statusInfoReadyEdge(CLK := NOT getRouterStatusInfo.bBusy AND NOT getRouterStatusInfo.bError);
IF (statusInfoReadyEdge.Q) THEN
	totalMem := DWORD_TO_DINT(statusInfo.maxMem) / IING.ONE_KBYTE;
	freeMem := DWORD_TO_DINT(statusInfo.maxMemAvail) / IING.ONE_KBYTE;
	FC_GetLogger().info(iData := FC_4strConcat(iStr1 := 'Memory usage (KB): ', iStr2 := DINT_TO_STRING(freeMem),
		iStr3 := ' / ', iStr4 := DINT_TO_STRING(totalMem)));
END_IF


// I believe it goes to error in livonia since no data coming from this one, check out and handle errors

END_FUNCTION_BLOCK

// ---- BASE/Misc/FB_OneCycleSignalTof.TcPOU
FUNCTION_BLOCK FB_OneCycleSignalTof		// Delays iSignal by 1 PLC cycle
VAR_INPUT
	iSignal:		BOOL;	// signal to be delayed
END_VAR
VAR_OUTPUT
	oSignal:		BOOL;	// 1 PLC cycle delayed signal
END_VAR
VAR
	fallingEdge:	F_TRIG;
END_VAR

fallingEdge(CLK := iSignal);
oSignal := iSignal OR fallingEdge.Q;

END_FUNCTION_BLOCK

// ---- BASE/Misc/FB_TofOnRtrig.TcPOU
FUNCTION_BLOCK FB_TofOnRtrig		// Monitors a signal (R_TRIG) and creates a TOF
VAR_INPUT
	iBool:		BOOL;	// Signal to be monitored
	iTime:		TIME;	// TOF time
END_VAR
VAR_OUTPUT
	oBool: 		BOOL;	// Set TRUE for iTime on a rising edge of iBool
END_VAR
VAR
	rtrig:		R_TRIG;
	tof:		TOF;
END_VAR

rtrig(CLK := iBool);
tof(IN := rtrig.Q, PT := iTime, Q => oBool);

END_FUNCTION_BLOCK

// ---- BASE/Misc/FC_GetLocalAmsNetId.TcPOU
FUNCTION FC_GetLocalAmsNetId : T_AmsNetId		// Returns the local AMS net id

FC_GetLocalAmsNetId := IING.localAmsNetId;

END_FUNCTION

// ---- BASE/Misc/FC_GetLocalHostName.TcPOU
FUNCTION FC_GetLocalHostName : T_MaxString	// Returns the local host name

FC_GetLocalHostName := IING.localHostName;

END_FUNCTION

// ---- BASE/Misc/FC_GetMax3Arg.TcPOU
FUNCTION FC_GetMax3Arg : REAL
VAR_INPUT
	iVal1:	REAL;
	iVal2:	REAL;
	iVal3:	REAL;
END_VAR
VAR
	maxVal:	REAL;
END_VAR

maxVal := MAX(iVal1, iVal2);
maxVal := MAX(maxVal, iVal3);

FC_GetMax3Arg := maxVal;

END_FUNCTION

// ---- BASE/Misc/FC_GetMax3Lreals.TcPOU
FUNCTION FC_GetMax3Lreals : LREAL		// Returns the maximum of specified values
VAR_INPUT
	iLreal1:	LREAL;
	iLreal2:	LREAL;
	iLreal3:	LREAL;
END_VAR

FC_GetMax3Lreals := MAX(iLreal1, iLreal2);
FC_GetMax3Lreals := MAX(FC_GetMax3Lreals, iLreal3);

END_FUNCTION

// ---- BASE/Misc/FC_GetMax4Arg.TcPOU
FUNCTION FC_GetMax4Arg : REAL
VAR_INPUT
	iVal1:	REAL;
	iVal2:	REAL;
	iVal3:	REAL;
	iVal4:	REAL;
END_VAR
VAR
	maxVal:	REAL;
END_VAR

maxVal := FC_GetMax3Arg(iVal1, iVal2, iVal3);
maxVal := MAX(maxVal, iVal4);

FC_GetMax4Arg := maxVal;

END_FUNCTION

// ---- BASE/Misc/FC_GetMin2Arg.TcPOU
FUNCTION FC_GetMin2Arg : REAL
VAR_INPUT
	iVal1:	REAL;		// Must not be zero
	iVal2:	REAL;
END_VAR
VAR
	minVal:	REAL;
END_VAR

minVal := iVal1;

IF (iVal2 <> 0) THEN
	minVal := MIN(minVal, iVal2);
END_IF

FC_GetMin2Arg := minVal;

END_FUNCTION

// ---- BASE/Misc/FC_GetMin3Arg.TcPOU
FUNCTION FC_GetMin3Arg : REAL
VAR_INPUT
	iVal1:	REAL;		// Must not be zero
	iVal2:	REAL;
	iVal3:	REAL;
END_VAR
VAR
	minVal:	REAL;
END_VAR

minVal := FC_GetMin2Arg(iVal1, iVal2);
minVal := FC_GetMin2Arg(minVal, iVal3);

FC_GetMin3Arg := minVal;

END_FUNCTION

// ---- BASE/Misc/FC_GetMin3Lreals.TcPOU
FUNCTION FC_GetMin3Lreals : LREAL		// Returns the minimum of specified values 
VAR_INPUT
	iLreal1:	LREAL;
	iLreal2:	LREAL;
	iLreal3:	LREAL;
END_VAR

FC_GetMin3Lreals := MIN(iLreal1, iLreal2);
FC_GetMin3Lreals := MIN(FC_GetMin3Lreals, iLreal3);

END_FUNCTION

// ---- BASE/Misc/FC_GetMin4Arg.TcPOU
FUNCTION FC_GetMin4Arg : REAL
VAR_INPUT
	iVal1:	REAL;		// Must not be zero
	iVal2:	REAL;
	iVal3:	REAL;
	iVal4:	REAL;
END_VAR
VAR
	minVal:	REAL;
END_VAR

minVal := FC_GetMin3Arg(iVal1, iVal2, iVal3);
minVal := FC_GetMin2Arg(minVal, iVal4);

FC_GetMin4Arg := minVal;

END_FUNCTION

// ---- BASE/NumberUtils/AddREAL.TcPOU
FUNCTION AddREAL : BOOL				// Increments the given UINT value
VAR_INPUT
	iAdd:	REAL;
END_VAR
VAR_IN_OUT
	ioNum:	REAL;		// Value to increment
END_VAR

ioNum := ioNum + iAdd;

END_FUNCTION

// ---- BASE/NumberUtils/DecINT.TcPOU
FUNCTION DecINT : INT				// Increments the given UINT value
VAR_IN_OUT
	ioNum:	INT;		// Value to increment
END_VAR

DecINT := ioNum := ioNum - 1;

END_FUNCTION

// ---- BASE/NumberUtils/FC_CheckMinMaxInt.TcPOU
FUNCTION FC_CheckMinMaxInt : INT	// Checks if the given value is within the min/max and if not will set either the MIN/MAX value
VAR_INPUT
	iValue:		INT;
	iMin:		INT;
	iMax:		int;
END_VAR

IF (iValue > iMax) THEN
	FC_CheckMinMaxInt := iMax;
ELSIF (iValue < iMin) THEN
	FC_CheckMinMaxInt := iMin;
ELSE
	FC_CheckMinMaxInt := iValue;
END_IF

END_FUNCTION

// ---- BASE/NumberUtils/FC_CheckMinMaxReal.TcPOU
FUNCTION FC_CheckMinMaxReal : REAL		// Checks if the given value is within the min/max and if not will set either the MIN/MAX value
VAR_INPUT
	iValue:		REAL;
	iMin:		REAL;
	iMax:		REAL;
END_VAR

IF (iValue > iMax) THEN
	FC_CheckMinMaxReal := iMax;
ELSIF (iValue < iMin) THEN
	FC_CheckMinMaxReal := iMin;
ELSE
	FC_CheckMinMaxReal := iValue;
END_IF

END_FUNCTION

// ---- BASE/NumberUtils/FC_KeepBetweenMinMax.TcPOU
FUNCTION FC_KeepBetweenMinMax : LREAL			// Keeps the given iValue in between iMin (Floor) and iMax (Ceiling)  
VAR_INPUT
	iValue:		LREAL;
	iMin:		LREAL;
	iMax:		LREAL;
END_VAR

IF (iValue > iMax) THEN
	FC_KeepBetweenMinMax := iMax;
ELSIF (iValue < iMin) THEN
	FC_KeepBetweenMinMax := iMin;
ELSE
	FC_KeepBetweenMinMax := iValue;
END_IF

END_FUNCTION

// ---- BASE/NumberUtils/FC_KeepBetweenMinMaxInt.TcPOU
FUNCTION FC_KeepBetweenMinMaxInt			// Keeps the given ioValue in between iMin (Floor) and iMax (Ceiling)  
VAR_INPUT
	iMin:		INT;
	iMax:		INT;
END_VAR
VAR_IN_OUT
	ioValue:		INT;
END_VAR

IF (ioValue > iMax) THEN
	ioValue := iMax;
ELSIF (ioValue < iMin) THEN
	ioValue := iMin;
END_IF

END_FUNCTION

// ---- BASE/NumberUtils/FC_KeepRealBetweenMinMax.TcPOU
FUNCTION FC_KeepRealBetweenMinMax : REAL			// Keeps the given iValue in between iMin (Floor) and iMax (Ceiling)  
VAR_INPUT
	iValue:		REAL;
	iMin:		REAL;
	iMax:		REAL;
END_VAR

IF (iValue > iMax) THEN
	FC_KeepRealBetweenMinMax := iMax;
ELSIF (iValue < iMin) THEN
	FC_KeepRealBetweenMinMax := iMin;
ELSE
	FC_KeepRealBetweenMinMax := iValue;
END_IF

END_FUNCTION

// ---- BASE/NumberUtils/FC_LimitMaxReal.TcPOU
FUNCTION FC_LimitMaxReal : bool
VAR_INPUT
	iMaster:		REAL;
END_VAR
VAR_IN_OUT
	ioSlave:		REAL;
END_VAR

IF (ioSlave > iMaster) THEN
	ioSlave := iMaster;
END_IF

END_FUNCTION

// ---- BASE/NumberUtils/FC_LimitMinReal.TcPOU
FUNCTION FC_LimitMinReal : bool
VAR_INPUT
	iMaster:	REAL;
END_VAR
VAR_IN_OUT
	ioSlave:		REAL;
END_VAR

IF (ioSlave < iMaster) THEN
	ioSlave := iMaster;
END_IF

END_FUNCTION

// ---- BASE/NumberUtils/FC_WithinMinMax.TcPOU
FUNCTION FC_WithinMinMax : BOOL		// Checks if the specified value is within the target range, returns TRUE if within range, FALSE otherwise
VAR_INPUT
	iValue:			LREAL;		// Value to be checked
	iMin:			LREAL;		// Target value
	iMax:			LREAL;		// This value is allowed below and above
END_VAR

FC_WithinMinMax := (iValue >= iMin) AND (iValue <= iMax);

END_FUNCTION

// ---- BASE/NumberUtils/FC_WithinRange.TcPOU
FUNCTION FC_WithinRange : BOOL		// Checks if the specified value is within the target range, returns TRUE if within range, FALSE otherwise
VAR_INPUT
	iValue:			LREAL;		// Value to be checked
	iTarget:		LREAL;		// Target value
	iRange:			LREAL;		// This value is allowed below and above
END_VAR
VAR
	minValue:	LREAL;
	maxValue:	LREAL;
END_VAR

minValue := iTarget - iRange;
maxValue := iTarget + iRange;
FC_WithinRange := (iValue >= minValue) AND (iValue <= maxValue);

END_FUNCTION

// ---- BASE/NumberUtils/IncINT.TcPOU
FUNCTION IncINT : INT				// Increments the given UINT value
VAR_IN_OUT
	ioNum:	INT;		// Value to increment
END_VAR

IncINT := ioNum := ioNum + 1;

END_FUNCTION

// ---- BASE/NumberUtils/IncUINT.TcPOU
FUNCTION IncUINT : UINT				// Increments the given UINT value
VAR_IN_OUT
	ioNum:	UINT;		// Value to increment
END_VAR

IncUINT := ioNum := ioNum + 1;

END_FUNCTION

// ---- BASE/NumberUtils/IncULINT.TcPOU
FUNCTION IncULINT : ULINT		// Increments the given ULINT value
VAR_IN_OUT
	ioNum:	ULINT;		// Value to increment
END_VAR

IncULINT := ioNum := ioNum + 1;

END_FUNCTION

// ---- BASE/Observer/FB_GenericObserver.TcPOU
FUNCTION_BLOCK ABSTRACT FB_GenericObserver		// To be extended by the REAL observer
VAR
	observers:		ARRAY[0..GVL_GENERIC_OBSERVER.OBSERVER_CNT-1] OF ST_GENERIC_OBSERVER;
	validObservers:	ST_VALID_OBSERVERS;
END_VAR

METHOD PUBLIC deregisterObserver : BOOL
VAR_INPUT
	iWho:				T_SHORT_STR;
END_VAR
VAR
	i: 					INT;
END_VAR
FOR i := 0 TO GVL_GENERIC_OBSERVER.OBSERVER_CNT-1 BY 1 DO
	IF (IsStringEqualIgnoreCase(observers[i].who, iWho)) THEN
		observers[i].who := IING.STRING_BLANK;
	END_IF
END_FOR
END_METHOD

METHOD PUBLIC getObservers : BOOL
VAR_INPUT
END_VAR
VAR
	i: 					INT;
END_VAR
validObservers.cnt := 0;
FOR i := 0 TO GVL_GENERIC_OBSERVER.OBSERVER_CNT-1 BY 1 DO
	IF (FC_StringNotEmpty(observers[i].who)) THEN
		validObservers.observers[validObservers.cnt].observer := observers[i].observer;
		IncInt(validObservers.cnt);
	END_IF
END_FOR
END_METHOD

METHOD PUBLIC registerObserver : BOOL
VAR_INPUT
	iWho:				T_SHORT_STR;
	iObserver:			POINTER TO BYTE;
END_VAR
VAR
	i: 					INT;
END_VAR
// Search if already registered, we do not want to register this twice
FOR i := 0 TO GVL_GENERIC_OBSERVER.OBSERVER_CNT-1 BY 1 DO
	IF (IsStringEqualIgnoreCase(observers[i].who, iWho)) THEN
		observers[i].observer := iObserver;	// Override the observer since it may have changed (re-initialised)
		RETURN;		
	END_IF
END_FOR

// Find 1st free element
FOR i := 0 TO GVL_GENERIC_OBSERVER.OBSERVER_CNT-1 BY 1 DO
	IF (FC_StringEmpty(observers[i].who)) THEN
		observers[i].observer := iObserver;
		observers[i].who := iWho;
		RETURN;		
	END_IF
END_FOR
END_METHOD

END_FUNCTION_BLOCK

// ---- BASE/StringUtils/IsStringEqualIgnoreCase.TcPOU
FUNCTION IsStringEqualIgnoreCase : BOOL
VAR_INPUT
	iString1:	STRING;
	iString2:	STRING;
END_VAR

IsStringEqualIgnoreCase := F_ToUCase(iString1) = F_ToUCase(iString2);

END_FUNCTION

// ---- BASE/StringUtils/FC_5strConcat.TcPOU
FUNCTION FC_5strConcat : T_DEFAULT_STR		// Concatenates 4 strings
VAR_INPUT
	iStr1:		T_DEFAULT_STR;
	iStr2:		T_DEFAULT_STR;
	iStr3:		T_DEFAULT_STR;
	iStr4:		T_DEFAULT_STR;
	iStr5:		T_DEFAULT_STR;
END_VAR

FC_5strConcat := CONCAT(FC_4strConcat(iStr1, iStr2, iStr3, iStr4),iStr5);

END_FUNCTION

// ---- BASE/StringUtils/FC_6strConcat.TcPOU
FUNCTION FC_6strConcat : T_DEFAULT_STR		// Concatenates 4 strings
VAR_INPUT
	iStr1:		T_DEFAULT_STR;
	iStr2:		T_DEFAULT_STR;
	iStr3:		T_DEFAULT_STR;
	iStr4:		T_DEFAULT_STR;
	iStr5:		T_DEFAULT_STR;
	iStr6:		T_DEFAULT_STR;
END_VAR

FC_6strConcat := CONCAT(FC_5strConcat(iStr1, iStr2, iStr3, iStr4, iStr5), iStr6);

END_FUNCTION

// ---- BASE/StringUtils/FC_6strConcatSeparator.TcPOU
FUNCTION FC_6strConcatSeparator : T_DEFAULT_STR		// Concatenates 5 strings with given separator
VAR_INPUT
	iSeparator:		STRING := IING.STRING_UNDERSCORE;
	iStr1:			T_DEFAULT_STR;
	iStr2:			T_DEFAULT_STR;
	iStr3:			T_DEFAULT_STR;
	iStr4:			T_DEFAULT_STR;
	iStr5:			T_DEFAULT_STR;
	iStr6:			T_DEFAULT_STR;
END_VAR

FC_6strConcatSeparator := FC_2strConcatSeparator(iSeparator := iSeparator,
	iStr1 := FC_5strConcatSeparator(iSeparator := iSeparator, iStr1 := iStr1, iStr2 := iStr2, iStr3 := iStr3, iStr4 := iStr4, iStr5 := iStr5), iStr2 := iStr6);

END_FUNCTION

// ---- BASE/StringUtils/FC_7strConcat.TcPOU
FUNCTION FC_7strConcat : T_DEFAULT_STR
VAR_INPUT
	iStr1:		T_DEFAULT_STR;
	iStr2:		T_DEFAULT_STR;
	iStr3:		T_DEFAULT_STR;
	iStr4:		T_DEFAULT_STR;
	iStr5:		T_DEFAULT_STR;
	iStr6:		T_DEFAULT_STR;
	iStr7:		T_DEFAULT_STR;
END_VAR

FC_7strConcat := CONCAT(FC_6strConcat(iStr1, iStr2, iStr3, iStr4, iStr5, iStr6), iStr7);

END_FUNCTION

// ---- BASE/StringUtils/FC_7strConcatSeparator.TcPOU
FUNCTION FC_7strConcatSeparator : T_DEFAULT_STR
VAR_INPUT
	iSeparator:		STRING := IING.STRING_UNDERSCORE;
	iStr1:			T_DEFAULT_STR;
	iStr2:			T_DEFAULT_STR;
	iStr3:			T_DEFAULT_STR;
	iStr4:			T_DEFAULT_STR;
	iStr5:			T_DEFAULT_STR;
	iStr6:			T_DEFAULT_STR;
	iStr7:			T_DEFAULT_STR;
END_VAR

FC_7strConcatSeparator := FC_2strConcatSeparator(iSeparator, FC_6strConcatSeparator(iSeparator, iStr1, iStr2, iStr3, iStr4, iStr5, iStr6), iStr7);

END_FUNCTION

// ---- BASE/StringUtils/FC_8strConcat.TcPOU
FUNCTION FC_8strConcat : T_DEFAULT_STR		// Concatenates 4 strings
VAR_INPUT
	iStr1:		T_DEFAULT_STR;
	iStr2:		T_DEFAULT_STR;
	iStr3:		T_DEFAULT_STR;
	iStr4:		T_DEFAULT_STR;
	iStr5:		T_DEFAULT_STR;
	iStr6:		T_DEFAULT_STR;
	iStr7:		T_DEFAULT_STR;
	iStr8:		T_DEFAULT_STR;
END_VAR

FC_8strConcat := CONCAT(FC_7strConcat(iStr1, iStr2, iStr3, iStr4, iStr5, iStr6, iStr7), iStr8);

END_FUNCTION

// ---- BASE/StringUtils/FC_8strConcatSeparator.TcPOU
FUNCTION FC_8strConcatSeparator : T_DEFAULT_STR
VAR_INPUT
	iSeparator:		STRING := IING.STRING_UNDERSCORE;
	iStr1:			T_DEFAULT_STR;
	iStr2:			T_DEFAULT_STR;
	iStr3:			T_DEFAULT_STR;
	iStr4:			T_DEFAULT_STR;
	iStr5:			T_DEFAULT_STR;
	iStr6:			T_DEFAULT_STR;
	iStr7:			T_DEFAULT_STR;
	iStr8:			T_DEFAULT_STR;
END_VAR

FC_8strConcatSeparator := FC_2strConcatSeparator(iSeparator, FC_7strConcatSeparator(iSeparator, iStr1, iStr2, iStr3, iStr4, iStr5, iStr6, iStr7), iStr8);

END_FUNCTION

// ---- BASE/StringUtils/FC_FindLastOccurence.TcPOU
FUNCTION FC_FindLastOccurence : INT		// Finds the last occurance of a character inside a string
VAR_INPUT
	iStr:			T_MaxString;		// String in where to search
	iStrTofind:		T_SHORT_STR;		// Character to search for
END_VAR
VAR
	i:			INT;
	pos:		INT;
	str:		T_MaxString;
	strLen:		INT;
END_VAR

// Example
// C:\Users\Administrator\Desktop\restartHmi.bat
//   3     9             23      31

FC_FindLastOccurence := 0;
str := iStr;
pos := FIND(str, iStrTofind);
WHILE (pos > 0)  DO
	strLen := LEN(str);
	pos := FIND(str, iStrTofind);
	str := MID(STR := str, LEN := strLen - pos, POS := pos + 1);
	FC_FindLastOccurence := FC_FindLastOccurence + pos;
END_WHILE

END_FUNCTION

// ---- BASE/StringUtils/FC_InitializeNameAsNeeded.TcPOU
FUNCTION FC_InitializeNameAsNeeded	// Can be used to initialize the given name of a component
VAR_INPUT
	iInit:	T_SHORT_STR;		// Initial value
END_VAR
VAR_IN_OUT
	ioMonitor:	T_SHORT_STR;	// String to be monitored
END_VAR

IF (NOT FC_IsBaseNameDefined(ioMonitor)) THEN
	ioMonitor := iInit;
END_IF

END_FUNCTION

// ---- BASE/StringUtils/FC_IsBaseNameDefined.TcPOU
FUNCTION FC_IsBaseNameDefined : bool
VAR_INPUT
	iName:	STRING;
END_VAR
VAR
	equalsNameHere:			BOOL;
	equalsQuestionMarks:	BOOL;
END_VAR

equalsQuestionMarks := IsStringEqualIgnoreCase(iName, IING.STRING_BASE_SETTINGS_INITIAL_NAME);
equalsNameHere := IsStringEqualIgnoreCase(iName, 'name here');

FC_IsBaseNameDefined := NOT equalsQuestionMarks AND NOT equalsNameHere AND FC_StringNotEmpty(iName);

END_FUNCTION

// ---- BASE/StringUtils/FC_LrealFormatter.TcPOU
FUNCTION FC_LrealFormatter : T_SHORT_STR
VAR_INPUT
	iLreal:				LREAL;
	iNumberOfDecimals:	INT;
END_VAR

FC_LrealFormatter := LREAL_TO_FMTSTR(in := iLreal, iPrecision := iNumberOfDecimals, bRound := FALSE);

END_FUNCTION

// ---- BASE/StringUtils/FC_RealFormatter.TcPOU
FUNCTION FC_RealFormatter : T_SHORT_STR
VAR_INPUT
	iReal:				REAL;
	iNumberOfDecimals:	INT;
END_VAR

FC_RealFormatter := LREAL_TO_FMTSTR(in := iReal, iPrecision := iNumberOfDecimals, bRound := FALSE);

END_FUNCTION

// ---- LOGGING/FileLogger/FB_FileLogger.TcPOU
FUNCTION_BLOCK FB_FileLogger IMPLEMENTS I_Logger				// File logger implementation
VAR_INPUT
	iAmsNetId:					T_AmsNetId := IING.STRING_BLANK;	// Where to write the file
	iPath:						T_DEFAULT_STR;					// Path where to log, this MAY NOT contain the file name
	iFileName:					T_SHORT_STR;					// File name for the log files, US style date will be prepended to the file name
END_VAR
VAR_OUTPUT
	oHmi:						ST_FILE_LOGGER_HMI;
END_VAR
VAR
	tcHmiCs:	TC_HMI_CS;	


	service:					ST_FILE_LOGGER_SERVICE;
	controlSignalsFb:			FB_ControlSignalsV2;
	
	
	currentFileNameAndPath:		FB_FileNameAndPath;
	fileWriter:					FB_FileWriterV2;
	
	stopWriting:				BOOL;							// Needed to we can rename the file
	fileScanner:				FB_FileScannerV2;
	higestNumberInFileName:		INT;
	
	newFileName:				T_SHORT_STR;
	newFileNameHelper:			FB_FileNameAndPath;
	fileRenamer:				FB_FileRename;
	fileRenameError:			UDINT;
	lastFileSize:				DINT;
	autoResetTimer:				TON;
	tracingTimer:				TON;
	
	stepChanged:				BOOL;
	step:						E_FILE_LOGGER_STEPS;
	oldStepForStepChangeOnly:	E_FILE_LOGGER_STEPS;			// Dont use for anything else
	prevStep:					E_FILE_LOGGER_STEPS;
	
	observerName:				STRING := 'fileLogger';
END_VAR
VAR PERSISTENT
	settings:					ST_FILE_LOGGER_SETTINGS;
	fileCnt:					INT := 0;
	initCalled:	 				INT;
	reInitCalled:				INT;
	exitCalled:					INT;
END_VAR

controlSignalsFb(iExternalReset := autoResetTimer.Q, ioTcHmi := tcHmiCs);
currentFileNameAndPath.setPathAndFileName(iPath := iPath, iFileName := FC_2strConcatSeparator(iSeparator := IING.STRING_UNDERSCORE, iStr1 := FC_GetUsDateString(), iStr2 := iFileName));

CASE step OF
	E_FILE_LOGGER_STEPS.WAIT_ACTIVITY:
		// When the file gets renamed, the fileSize from the writer gets updated ONLY after the next file write, here we ensure we dont start renaming instantly after the previous rename  
		gotoNextStep(iCondition := fileWriter.oFileSize <> lastFileSize, iNextStep := E_FILE_LOGGER_STEPS.CHECK_SIZE);
	
	E_FILE_LOGGER_STEPS.CHECK_SIZE:
		gotoNextStep(iCondition := (fileWriter.oFileSize > settings.MaxFileSizeMB * IING.ONE_MBYTE), iNextStep := E_FILE_LOGGER_STEPS.CLOSE_FILE);
	
	E_FILE_LOGGER_STEPS.CLOSE_FILE:
		gotoNextStep(iCondition := fileWriter.oFileClosed, iNextStep := E_FILE_LOGGER_STEPS.SCAN_FOLDER);
	
	E_FILE_LOGGER_STEPS.SCAN_FOLDER:
		gotoNextStep(iCondition := fileScanner.oDone, iNextStep := E_FILE_LOGGER_STEPS.ITERATE_FILES);
	
	E_FILE_LOGGER_STEPS.ITERATE_FILES:
		higestNumberInFileName := iterateFiles(iBaseName := currentFileNameAndPath.getFileNameWithExtension(),
			iScannedFiles := ADR(fileScanner.oFiles), iNumberOfFiles := fileScanner.oFilesFound);
	
		gotoNextStep(iCondition := TRUE, iNextStep := E_FILE_LOGGER_STEPS.RENAME_FILE);

	E_FILE_LOGGER_STEPS.RENAME_FILE:
		gotoNextStep(iCondition := fileRenamer.bError, iNextStep := E_FILE_LOGGER_STEPS.RENAME_FILE_ERROR);
		gotoNextStep(iCondition := NOT fileRenamer.bBusy, iNextStep := E_FILE_LOGGER_STEPS.WAIT_ACTIVITY);
		
	E_FILE_LOGGER_STEPS.RENAME_FILE_ERROR:
		gotoNextStep(iCondition := controlSignalsFb.oControlSignals^.out.resetPulse, iNextStep := E_FILE_LOGGER_STEPS.CHECK_SIZE);
ELSE
	step := E_FILE_LOGGER_STEPS.WAIT_ACTIVITY;
END_CASE
updateOldStep();

// For rename to succeed, the log file is first to be closed, when rename fails, we let the logging continue hence that step is not included here
// One thing to notice is that when doLog is called while file rename is ongoing, the file writer will automatically buffer the data and write to file as soon as renaming is completed
stopWriting := (step = E_FILE_LOGGER_STEPS.CLOSE_FILE) OR (step = E_FILE_LOGGER_STEPS.SCAN_FOLDER) OR (step = E_FILE_LOGGER_STEPS.ITERATE_FILES) OR (step = E_FILE_LOGGER_STEPS.RENAME_FILE);

fileWriter(iKeepFileOpen := TRUE, iAmsNetId := iAmsNetId, iFileNameAndPath := currentFileNameAndPath.getFileNameAndPath(), iFlush := service.doFileFlush, iStopWriting := stopWriting,
	iControlSignals := controlSignalsFb.oControlSignals^.out, oFileWriterRecordCnt => oHmi.fileWriterRecordCnt, oFileWriterBytesUsed => oHmi.fileWriterBytesUsed);

fileScanner(iAmsNetId := iAmsNetId, iPath := iPath, iFileName := currentFileNameAndPath.getFileNameWithExtension(),
	iScan := (step = E_FILE_LOGGER_STEPS.SCAN_FOLDER) OR (step = E_FILE_LOGGER_STEPS.ITERATE_FILES), iControlSignals := controlSignalsFb.oControlSignals^.out);

IF (stepChanged AND (step = (E_FILE_LOGGER_STEPS.RENAME_FILE))) THEN
	lastFileSize := fileWriter.oFileSize;
	newFileName := CONCAT(STR1 := currentFileNameAndPath.getFileNameNoExtension(), STR2 := INT_TO_STRING(higestNumberInFileName + 1));
	newFileNameHelper.setPath_FileNameAndExtension(iPath := iPath, iFileName := newFileName, iExtension := currentFileNameAndPath.getExtension());
END_IF	

fileRenamer(sNetId := iAmsNetId, sOldName := currentFileNameAndPath.getFileNameAndPath(), sNewName := newFileNameHelper.getFileNameAndPath(), ePath := E_OpenPath.PATH_GENERIC,
	bExecute := (step = E_FILE_LOGGER_STEPS.RENAME_FILE), tTimeout := IING.ADS_WRITE_TIMEOUT, nErrID => fileRenameError);

autoSwitchOffTracing();
autoReset();
hmi();

METHOD autoReset : BOOL
autoResetTimer(IN := oHmi.error, PT := settings.autoResetTime);
END_METHOD

METHOD PRIVATE autoSwitchOffTracing : BOOL	// Tracing can create a lot of file writing and load, therefore we switch this off after a while
oHmi.tracingOn := settings.logLevel = E_LOG_LEVEL.TRACE;

tracingTimer(IN := settings.enableMaxTracingTime AND oHmi.tracingOn, PT := settings.maxTracingTime, ET => oHmi.tracingTimeExpired);
IF (tracingTimer.Q) THEN
	settings.logLevel := E_LOG_LEVEL.ERROR;
END_IF
END_METHOD

METHOD PUBLIC debug : BOOL	// Logs the data with log level 'DEBUG'
VAR_INPUT
	iData:		T_DEFAULT_STR;						// Data to be logged, limited to 255 characters
END_VAR
doLog(iData := iData, iLevel := E_LOG_LEVEL.DEBUG);
END_METHOD

METHOD PUBLIC deregister : BOOL
VAR_INPUT
	iWho:				T_SHORT_STR;
END_VAR
END_METHOD

METHOD PUBLIC doLog : BOOL		// Logs the data to the file (depending on the activated log level)
								// Timestamp is always added in front of the data
VAR_INPUT
	iData:					T_DEFAULT_STR;						// Data to be logged, limited to 255 characters
	iLevel:					E_LOG_LEVEL := E_LOG_LEVEL.ERROR;	// Log level
END_VAR
VAR
	logLevel:				FB_LogLevel;
	header:					T_DEFAULT_STR;
	fullLine:				T_LONG_STR_512;
	
	runningNumberAsString:	T_SHORT_STR;
	eventIdAsString:		T_SHORT_STR;
	
	testSuccess: 			BOOL;
END_VAR
(*
v: Visible
						doLog called with
						-----------------
						ERROR		WARN		INFO		DEBUG		TRACE
Current log level
-----------------
OFF						
ERROR					v
WARN					v			v
INFO					v			v			v
DEBUG					v			v			v			v
TRACE					v			v			v			v			v
*)

// Logging is only done when the log level is higher or equal the current log level
IF (iLevel >= settings.logLevel) THEN
	logLevel.set(iLevel);

	header := FC_2strConcatSeparator (iSeparator := IING.STRING_SPACE, iStr1 := FC_GetLocalDateAndTimeString(), iStr2 := logLevel.asString());
	
	
	// iData can be up to 255 chars, including the header therefore more than 255, we use CONCAT2 and 'long' string 
	fullLine := CONCAT(STR1 := header, STR2 := IING.STRING_SPACE);
	testSuccess := CONCAT2(pSrcString1  := ADR(fullLine), pSrcString2 := ADR(iData), pDstString := ADR(fullLine), nDstSize := SIZEOF(fullLine));
	testSuccess := CONCAT2(pSrcString1  := ADR(fullLine), pSrcString2 := ADR(IING.STRING_LINE_FEED), pDstString := ADR(fullLine), nDstSize := SIZEOF(fullLine));
	
	fileWriter.doWrite(fullLine);
END_IF

// Just in case something went wrong and the level is not within the enum range
IF (settings.logLevel > E_LOG_LEVEL.OFF) THEN
	settings.logLevel := E_LOG_LEVEL.ERROR;
END_IF
END_METHOD

METHOD PUBLIC error : BOOL	// Logs the data with log level 'ERROR'
VAR_INPUT
	iData:		T_DEFAULT_STR;						// Data to be logged, limited to 255 characters
END_VAR
doLog(iData := iData, iLevel := E_LOG_LEVEL.ERROR);
END_METHOD

METHOD FB_exit : BOOL
VAR_INPUT
	bInCopyCode : BOOL; // if TRUE, the exit method is called for exiting an instance that is copied afterwards (online change).
END_VAR
IncInt(exitCalled);

//FC_GetLogger().deregister(observerName);
END_METHOD

METHOD FB_init : BOOL
VAR_INPUT
	bInitRetains : BOOL; // if TRUE, the retain variables are initialized (warm start / cold start)
	bInCopyCode : BOOL;  // if TRUE, the instance afterwards gets moved into the copy code (online change)
END_VAR
IncInt(initCalled);

//FC_GetLogger().register(observerName, THIS^);
END_METHOD

METHOD FB_reinit : BOOL
IncInt(reInitCalled);

//FC_GetLogger().register(observerName, THIS^);
END_METHOD

METHOD PRIVATE gotoNextStep : BOOL
VAR_INPUT
	iCondition:	BOOL;
	iNextStep:	E_FILE_LOGGER_STEPS;
END_VAR
IF (NOT (step<>oldStepForStepChangeOnly)) THEN
	IF (iCondition) THEN
		step := iNextStep;
	END_IF
END_IF
END_METHOD

METHOD PRIVATE hmi : BOOL
oHmi.service REF= service;
oHmi.settings REF= settings;
oHmi.controlSignals REF= controlSignalsFb.oControlSignals^.in;

IF (step = E_FILE_LOGGER_STEPS.SCAN_FOLDER) THEN
	oHmi.error := fileScanner.oError;
	oHmi.adsErrorCode := fileScanner.oAdsErrorCode;
ELSIF (step = E_FILE_LOGGER_STEPS.RENAME_FILE_ERROR) THEN
	oHmi.error := TRUE;	
	oHmi.adsErrorCode := FC_GetAdsErrorCode(fileRenameError);				
ELSE
	oHmi.error := fileWriter.oError;
	oHmi.adsErrorCode := fileWriter.oAdsErrorCode;
END_IF
	
oHmi.amsNetId := iAmsNetId;
oHmi.fileNameAndPath := currentFileNameAndPath.getFileNameAndPath();

oHmi.fileWriterOverflowCount := fileWriter.oOverflowCount;

// Found from autoSwitchOffTracing
//oHmi.tracingOn 
//oHmi.tracingTimeLeft
END_METHOD

METHOD PUBLIC info : BOOL	// Logs the data with log level 'INFO'
VAR_INPUT
	iData:		T_DEFAULT_STR;						// Data to be logged, limited to 255 characters
END_VAR
doLog(iData := iData, iLevel := E_LOG_LEVEL.INFO);
END_METHOD

METHOD PRIVATE iterateFiles : INT		// Iterates the given files and stores the highest number as appended in the base file name
VAR_INPUT
	iBaseName:				T_SHORT_STR;				// Base name, eg. 2019-11-14-logging
	iScannedFiles:			POINTER TO T_SHORT_STR;		// Array of files as given by FB_FileScanner matching the base name
	iNumberOfFiles:			INT;						// Number of files in the scannedFiles array
END_VAR
VAR 
	i:						INT;						// For loop
	baseNameHelper:			FB_FileNameAndPath;
	scannedFileHelper:		FB_FileNameAndPath;
	fileNumberAsString:		T_SHORT_STR;
	fileNumber:				INT;
END_VAR
// Iterates the given files and stores the highest number as appended in the base file name, in this example it would be 3
// 2019-11-14-logging1.txt
// 2019-11-14-logging2.txt
// 2019-11-14-logging3.txt
baseNameHelper.setPathAndFileName(iPath := iPath, iFileName := iBaseName);

FOR i := 0 TO iNumberOfFiles -1 BY 1 DO
	scannedFileHelper.setPathAndFileName(iPath := iPath, iFileName := iScannedFiles[i]);
	fileNumberAsString := RIGHT(STR := scannedFileHelper.getFileNameNoExtension(), SIZE := LEN(scannedFileHelper.getFileNameNoExtension()) - LEN(baseNameHelper.getFileNameNoExtension()));
	
	fileNumber := STRING_TO_INT(fileNumberAsString);// If this fails, 0 will be returned so this is safe to do
	iterateFiles := MAX(fileNumber, iterateFiles);
END_FOR
END_METHOD

METHOD PUBLIC register : BOOL
VAR_INPUT
	iWho:		T_SHORT_STR;
	iObserver:	I_Logger;
END_VAR
END_METHOD

METHOD PUBLIC trace : BOOL	// Logs the data with log level 'TRACE'
VAR_INPUT
	iData:		T_DEFAULT_STR;						// Data to be logged, limited to 255 characters
END_VAR
doLog(iData := iData, iLevel := E_LOG_LEVEL.TRACE);
END_METHOD

ACTION updateOldStep:
IF (step <> oldStepForStepChangeOnly) THEN
	stepChanged := TRUE;
	prevStep := oldStepForStepChangeOnly;			// Otherwise next SWITCH CASE checks oldStep which was just updated here!!
	oldStepForStepChangeOnly := step;
ELSE 
	stepChanged := FALSE;
END_IF
END_ACTION

METHOD PUBLIC warn : BOOL	// Logs the data with log level 'WARN'
VAR_INPUT
	iData:		T_DEFAULT_STR;						// Data to be logged, limited to 255 characters
END_VAR
doLog(iData := iData, iLevel := E_LOG_LEVEL.WARN);
END_METHOD

END_FUNCTION_BLOCK

// ---- LOGGING/FileLogger/FB_FileNameAndPath.TcPOU
FUNCTION_BLOCK FB_FileNameAndPath		// Utility function for making file path/naming easier
VAR
	path:				T_DEFAULT_STR;
	fileName:			T_DEFAULT_STR;
	extension:			T_SHORT_STR;
	fileNameAndPath:	T_DEFAULT_STR;
END_VAR

METHOD public getExtension : T_SHORT_STR		// Returns the file extension
getExtension := extension;
END_METHOD

METHOD PUBLIC getFileNameAndPath : T_DEFAULT_STR		// Returns the full file name and path (including extension)
getFileNameAndPath := fileNameAndPath;
END_METHOD

METHOD public getFileNameNoExtension : T_DEFAULT_STR		// Returns the file name without the extension
getFileNameNoExtension := fileName;
END_METHOD

METHOD PUBLIC getFileNameWithExtension : T_DEFAULT_STR	// Returns the file name with extension
getFileNameWithExtension := FC_2strConcatSeparator(iSeparator := IING.STRING_DOT, iStr1 := fileName, iStr2 := extension);
END_METHOD

METHOD PUBLIC getPath : T_DEFAULT_STR		// Returns the file path
getPath := path;
END_METHOD

METHOD PUBLIC setPath_FileNameAndExtension : BOOL	// Setter for file name, extension and path
VAR_INPUT
	iPath:			T_DEFAULT_STR;		// Path
	iFileName:		T_SHORT_STR;		// File name excluding the extension
	iExtension:		T_SHORT_STR;		// The file extension
END_VAR
setPathAndFileName(iPath := iPath, iFileName := FC_3strConcat(iStr1 := iFileName, iStr2 := IING.STRING_DOT, iStr3 := iExtension));
END_METHOD

METHOD public setPathAndFileName : BOOL		// Setter for file name (including extension) and path
VAR_INPUT
	iPath:			T_DEFAULT_STR;		// Path
	iFileName:		T_SHORT_STR;		// File name including the extension
END_VAR

VAR
	dotPos:int;
END_VAR
// Construct path having back slash at the end
IF (RIGHT(iPath, 1) = IING.STRING_BACKSLASH) THEN
	path := iPath;
ELSE
	path := CONCAT(iPath, IING.STRING_BACKSLASH);
END_IF

// Construct file name with extension
dotPos := FIND(iFileName, IING.STRING_DOT);
IF (dotPos > 0) THEN
	fileName := LEFT(STR := iFileName, SIZE := dotPos -1);
	extension := RIGHT(STR := iFileName, SIZE := LEN(iFileName) - dotPos);
ELSE
	fileName := iFileName;
	extension := 'missing';
END_IF


fileNameAndPath := CONCAT(path, getFileNameWithExtension());
END_METHOD

END_FUNCTION_BLOCK

// ---- LOGGING/FileLogger/FB_FileWriterV2.TcPOU
FUNCTION_BLOCK FB_FileWriterV2	// Handles writing of lines to a file.  Maximum line length is 256 characters.
VAR_INPUT
	iKeepFileOpen:					BOOL;							// Set TRUE to keep the file open in between writes
	iAmsNetId:						T_AmsNetId := IING.STRING_BLANK;	// Where to write the file
	iFileNameAndPath:				T_DEFAULT_STR;					// File name and path of the file
	iFlush:							BOOL;							// Set TRUE when a file flush is needed (will actually close and re-open the file)
	iStopWriting:					BOOL;							// Used when the caller of this FB wants to temporarily stop writing (eg. when file rename is ongoing)
	iControlSignals:				ST_CONTROL_SIGNALS_OUT;			// Control signals (carrying reset signal)
END_VAR
VAR_OUTPUT
	oFileClosed:					BOOL;
	oFileSize:						DINT;
	oError:							BOOL;							// TRUE if a file writing error occurs
	oAdsErrorCode:					E_ADS_ERRORS;
	oOverflowCount:					UDINT;							// How many times we were not able to write all data to the file (due to internal memory constraints)
	
	oFileWriterRecordCnt:			UDINT;
	oFileWriterBytesUsed:			UDINT;
END_VAR
VAR
	fileHandle:						UINT := 0;
	fileHandleFromFB_FileOpen:		UINT := 0;						// Separate var since overwritten from FB_FileOpen even if not open anymore
	fileOpen:						FB_FileOpen;
	fileWrite:						FB_FileWrite;					// Not using FB_FilePuts since it is limited of writing T_MaxString
	fileClose:						FB_FileClose;

	fileTell:						FB_FileTell;
	
	dataToBeWritten:				BOOL;		// Helper to know when data is buffered and to be written
	
	fileNameCopy:					T_DEFAULT_STR;
	fileNameChangeEdge:				R_TRIG;
	flush:							BOOL;
	
	stepChanged:					BOOL;
	step:							E_FILE_WRITER_STEPS;
	oldStepForStepChangeOnly:		E_FILE_WRITER_STEPS;			// Dont use for anything else
	prevStep:						E_FILE_WRITER_STEPS;
	
	ringBufferMemory:				ARRAY[0..RINGBUFFER_SIZE_IN_BYTES-1] OF BYTE;
	ringBuffer:						FB_MemRingBuffer;
	
	longString:						STRING(LONGSTRING_SIZE_IN_BYTES);	// LEN2 has a restriction to 10000 chars
	
	fileOpeningError:				UDINT;
	fileWritingError:				UDINT;
	fileTellError:					UDINT;
	fileClosingError:				UDINT;
	
	bytesWritten:					UDINT;
END_VAR
VAR PERSISTENT
	overFlowCnt:					UDINT;	// Number of times overflow would have happened
	concatFailure:					UDINT;	// Number of concat failures, should stay at 0
END_VAR
VAR CONSTANT
	RINGBUFFER_SIZE_IN_BYTES:		UDINT := 30000;
	LONGSTRING_SIZE_IN_BYTES:		UDINT := 10000;
END_VAR

// When file name changes (eg. from logger), we need to close and re-open the file (with different name)
fileNameChangeEdge(CLK := NOT (iFileNameAndPath = fileNameCopy));
fileNameCopy := iFileNameAndPath;

IF (fileNameChangeEdge.Q OR iFlush) THEN		// Rising edge can easily get lost while writing is ongoing (can take several PLC cycles), therefore must 'save' it
	flush := TRUE;	
END_IF

dataToBeWritten := ringBuffer.nCount > 0;	// See doWrite

CASE step OF
	E_FILE_WRITER_STEPS.IDLE:
		gotoNextStep(iCondition := NOT iStopWriting AND iKeepFileOpen, iNextStep := E_FILE_WRITER_STEPS.OPEN_FILE);
		gotoNextStep(iCondition := NOT iStopWriting AND NOT iKeepFileOpen AND dataToBeWritten, iNextStep := E_FILE_WRITER_STEPS.OPEN_FILE);
		
	E_FILE_WRITER_STEPS.OPEN_FILE:
		gotoNextStep(iCondition := fileOpen.bError, iNextStep := E_FILE_WRITER_STEPS.OPENING_ERROR);
		gotoNextStep(iCondition := NOT fileOpen.bBusy, iNextStep := E_FILE_WRITER_STEPS.WAIT_DATA);
	
	E_FILE_WRITER_STEPS.WAIT_DATA:
		gotoNextStep(iCondition := dataToBeWritten, iNextStep := E_FILE_WRITER_STEPS.WRITE_LINE);
		gotoNextStep(iCondition := flush OR NOT iKeepFileOpen OR iStopWriting, iNextStep := E_FILE_WRITER_STEPS.CLOSE_FILE);

	E_FILE_WRITER_STEPS.WRITE_LINE:
		gotoNextStep(iCondition := fileWrite.bError, iNextStep := E_FILE_WRITER_STEPS.WRITING_ERROR);
		gotoNextStep(iCondition := NOT fileWrite.bBusy , iNextStep := E_FILE_WRITER_STEPS.CHECK_FILE);
		
	E_FILE_WRITER_STEPS.CHECK_FILE:
		gotoNextStep(iCondition := fileTell.bError, iNextStep := E_FILE_WRITER_STEPS.TELL_ERROR);
		gotoNextStep(iCondition := NOT fileTell.bBusy AND (flush OR iStopWriting OR NOT iKeepFileOpen), iNextStep := E_FILE_WRITER_STEPS.CLOSE_FILE);
		gotoNextStep(iCondition := NOT fileTell.bBusy, iNextStep := E_FILE_WRITER_STEPS.WAIT_DATA);

	E_FILE_WRITER_STEPS.CLOSE_FILE:
		flush := FALSE;
		gotoNextStep(iCondition := fileClose.bError, iNextStep := E_FILE_WRITER_STEPS.CLOSING_ERROR);
		gotoNextStep(iCondition := NOT fileClose.bBusy, iNextStep := E_FILE_WRITER_STEPS.CLEANUP);
	
	E_FILE_WRITER_STEPS.CLEANUP:
		fileHandle := 0;
		gotoNextStep(iCondition := TRUE, iNextStep := E_FILE_WRITER_STEPS.IDLE);
	
	E_FILE_WRITER_STEPS.OPENING_ERROR:
		oAdsErrorCode := FC_GetAdsErrorCode(fileOpeningError);
		gotoNextStep(iCondition := fileHandle <> 0, iNextStep := E_FILE_WRITER_STEPS.CLOSE_FILE);
		gotoNextStep(iCondition := iControlSignals.resetPulse, iNextStep := E_FILE_WRITER_STEPS.IDLE);

	E_FILE_WRITER_STEPS.WRITING_ERROR:
		oAdsErrorCode := FC_GetAdsErrorCode(fileWritingError);
		gotoNextStep(iCondition := fileHandle <> 0, iNextStep := E_FILE_WRITER_STEPS.CLOSE_FILE);
		gotoNextStep(iCondition := iControlSignals.resetPulse, iNextStep := E_FILE_WRITER_STEPS.IDLE);

	E_FILE_WRITER_STEPS.TELL_ERROR:
		oAdsErrorCode := FC_GetAdsErrorCode(fileTellError);
 		gotoNextStep(iCondition := fileHandle <> 0, iNextStep := E_FILE_WRITER_STEPS.CLOSE_FILE);
		gotoNextStep(iCondition := iControlSignals.resetPulse, iNextStep := E_FILE_WRITER_STEPS.IDLE);
		
	E_FILE_WRITER_STEPS.CLOSING_ERROR:
		oAdsErrorCode := FC_GetAdsErrorCode(fileClosingError);
		gotoNextStep(iCondition := iControlSignals.resetPulse, iNextStep := E_FILE_WRITER_STEPS.IDLE);
ELSE
	step := E_FILE_WRITER_STEPS.IDLE;
END_CASE
updateOldStep();


IF (stepChanged AND (step = E_FILE_WRITER_STEPS.WAIT_DATA) AND (prevStep = E_FILE_WRITER_STEPS.OPEN_FILE)) THEN
	fileHandle := fileHandleFromFB_FileOpen;
END_IF

fileOpen(sNetId := iAmsNetId, sPathName := iFileNameAndPath, nMode := FOPEN_MODEAPPEND,
	ePath := PATH_GENERIC, bExecute := (step = E_FILE_WRITER_STEPS.OPEN_FILE), hFile => fileHandleFromFB_FileOpen, tTimeout := IING.ADS_WRITE_TIMEOUT, nErrID => fileOpeningError);
	
// The data must be updated before the writing starts
concatBuffers(stepChanged AND (step = E_FILE_WRITER_STEPS.WRITE_LINE));	// Concatenates all data into a long string so writing is more efficient

fileWrite(sNetId := iAmsNetId, hFile := fileHandle, pWriteBuff := ADR(longString), cbWriteLen := LEN2(ADR(longString)), bExecute := (step = (E_FILE_WRITER_STEPS.WRITE_LINE)),
	tTimeout := IING.ADS_WRITE_TIMEOUT, nErrId => fileWritingError, cbWrite => bytesWritten);
	
fileTell(sNetId := iAmsNetId, hFile := fileHandle, bExecute := (step = E_FILE_WRITER_STEPS.CHECK_FILE), tTimeout := IING.ADS_WRITE_TIMEOUT, nSeekPos => oFileSize,
	nErrId => fileTellError);	
	
fileClose(sNetId := iAmsNetId, hFile := fileHandle, bExecute := (step = (E_FILE_WRITER_STEPS.CLOSE_FILE)), tTimeout := IING.ADS_WRITE_TIMEOUT, nErrId => fileClosingError);

ringBuffer(nCount => oFileWriterRecordCnt, cbSize => oFileWriterBytesUsed);

oFileClosed := (step = E_FILE_WRITER_STEPS.IDLE);		// In idle we can be sure the file is closed
oError := (step = E_FILE_WRITER_STEPS.OPENING_ERROR) OR (step = E_FILE_WRITER_STEPS.WRITING_ERROR) OR (step = E_FILE_WRITER_STEPS.CLOSING_ERROR);
oOverflowCount := overFlowCnt;

IF (iControlSignals.hardResetPulse) THEN
	step := E_FILE_WRITER_STEPS.IDLE;
	ringBuffer.A_Reset();
	flush := FALSE;
END_IF

METHOD PRIVATE concatBuffers : BOOL
VAR_INPUT
	iCondition:			BOOL;
END_VAR
VAR
	bufferedLine:		T_LONG_STR_512;	// Data read back from the ringBuffer, must be as big as iData in the doWrite method!
	trash:				T_LONG_STR_512;	// Must be as big as iData in the doWrite method!
	shouldFit:			BOOL;
	
	bufferedLineLen:	UDINT;
	longStringLen:		UDINT;
END_VAR
IF (iCondition) THEN
	longString := '';
	shouldFit := TRUE;
	WHILE (ringBuffer.nCount > 0 AND shouldFit) DO
		// We get the data but dont delete it yet
		ringBuffer.A_GetHead(pRead := ADR(bufferedLine), cbRead := SIZEOF(bufferedLine), pBuffer := ADR(ringBufferMemory), cbBuffer	:= SIZEOF(ringBufferMemory));

		// Check if bufferedLine will fit to longString
		bufferedLineLen := LEN2(ADR(bufferedLine));
		longStringLen:= LEN2(ADR(longString));
		shouldFit := (longStringLen + bufferedLineLen <= LONGSTRING_SIZE_IN_BYTES);	// Same size as longString
		IF (shouldFit) THEN
			// Here we concat onto longString, this should always succeed
			// If data would be too big for CONCAT2, that data that fits would be added and the rest discarded, therefore we check before hand to ensure all data gets logged correctly
			shouldFit := CONCAT2(pSrcString1  := ADR(longString), pSrcString2 := ADR(bufferedLine), pDstString := ADR(longString), nDstSize := SIZEOF(longString));
			IF (shouldFit) THEN
				// When the data did fit, we remove it from the ringBuffer (we read into a trash variable)
				ringBuffer.A_RemoveHead(pRead := ADR(trash), cbRead := SIZEOF(trash), pBuffer := ADR(ringBufferMemory), cbBuffer	:= SIZEOF(ringBufferMemory));
			ELSE
				// Should never come here
				IncUDINT(concatFailure); 
			END_IF
		ELSE
			;	// Its ok to leave the while loop since we will write (to file) all we got into longString, after that we create another longString and write again
			// The 10000 limitation means our file write, writes mostly 10000 bytes at a time
		END_IF
	END_WHILE
END_IF
END_METHOD

METHOD PUBLIC doWrite : BOOL		// Will add this data to the queue that will be written in the current PLC cycle.  Data is buffered and file write happens at most once/PLC cycle.
VAR_INPUT
	iData:		T_LONG_STR_512;		// The data to be written, up to 512 chars
END_VAR
// Add data to the FIFO

// If SIZEOF is used on iData, the ringbuffer always has entries that are as big as iData, even though the string would be 1 char only
// When using, LEN2, we can fit more data to the ringbuffer since rarely the iData will be the max length
// +1 is to account for the string variables final null (it is required!)
ringBuffer.A_AddTail(pWrite := ADR(iData), cbWrite := (LEN2(ADR(iData)) + 1), 							// What to write
					 pBuffer := ADR(ringBufferMemory), cbBuffer := SIZEOF(ringBufferMemory));	// The ringbuffer's memory	
					 
// If data doesnt fit anymore, bOk will be FALSE					 
IF (NOT ringBuffer.bOk) THEN
	IncUDINT(overflowCnt);	// More data is to be written in this PLC cycle but it doesnt fit the ringBuffer
END_IF
END_METHOD

METHOD PRIVATE gotoNextStep : BOOL
VAR_INPUT
	iCondition:	BOOL;
	iNextStep:	E_FILE_WRITER_STEPS;
END_VAR
IF (NOT (step<>oldStepForStepChangeOnly)) THEN
	IF (iCondition) THEN
		step := iNextStep;
	END_IF
END_IF
END_METHOD

ACTION updateOldStep:
IF (step <> oldStepForStepChangeOnly) THEN
	stepChanged := TRUE;
	prevStep := oldStepForStepChangeOnly;			// Otherwise next SWITCH CASE checks oldStep which was just updated here!!
	oldStepForStepChangeOnly := step;
ELSE 
	stepChanged := FALSE;
END_IF
END_ACTION

END_FUNCTION_BLOCK

// ---- LOGGING/FileLogger/FB_FileScannerV2.TcPOU
FUNCTION_BLOCK FB_FileScannerV2	// Scans the given folder for files with given name
VAR_INPUT
	iAmsNetId:					T_AmsNetId := IING.STRING_BLANK;	// Where to scan for files
	iPath:						T_DEFAULT_STR;					// Path where to scan, this MAY NOT contain the file name
	iFileName:					T_SHORT_STR;					// File names to match, do not include wildcards here
	iScan:						BOOL;							// TRUE will start the scanning
	iControlSignals:			ST_CONTROL_SIGNALS_OUT;			// Control signals (carrying reset signal)
END_VAR
VAR_OUTPUT
	oDone:						BOOL;									// Set TRUE when scanning is completed
	oFiles:						ARRAY[0..MAX_FILES-1] OF T_SHORT_STR;	// List of scanned files matching the given fileName
	oFilesFound:				INT;									// Number of matching files
	oError:						BOOL;									// Set TRUE when a scan error occurs
	oAdsErrorCode:				E_ADS_ERRORS;							// The error code in case oError is TRUE
END_VAR
VAR
	fileNameAndPath:			FB_FileNameAndPath;
	fileCnt:					INT;
	fileToSearch:				T_DEFAULT_STR;
	scanCommand:				E_EnumCmdType;
	scanFolder:					FB_EnumFindFileEntry;
	scanFolderError:			UDINT;

	stepChanged:				BOOL;
	step:						E_FILE_SCANNER_STEPS;
	oldStepForStepChangeOnly:	E_FILE_SCANNER_STEPS;			// Dont use for anything else
	prevStep:					E_FILE_SCANNER_STEPS;
END_VAR
VAR CONSTANT
	MAX_FILES:					INT := 100;
END_VAR

CASE step OF
	E_FILE_SCANNER_STEPS.IDLE:
		gotoNextStep(iCondition := iScan, iNextStep := E_FILE_SCANNER_STEPS.SCAN);
	
	E_FILE_SCANNER_STEPS.SCAN:
		gotoNextStep(iCondition := scanFolder.bError, iNextStep := E_FILE_SCANNER_STEPS.ERROR);
		gotoNextStep(iCondition := NOT scanFolder.bBusy, iNextStep := E_FILE_SCANNER_STEPS.STORE_FILE);	

	E_FILE_SCANNER_STEPS.STORE_FILE:
		IF (NOT scanFolder.bEOE) THEN
			IF (fileCnt < MAX_FILES) THEN
				oFiles[fileCnt] := scanFolder.stFindFile.sFileName;
				IncINT(fileCnt);
			END_IF
			gotoNextStep(iCondition := TRUE, iNextStep := E_FILE_SCANNER_STEPS.SCAN);		
		ELSE
			gotoNextStep(iCondition := TRUE, iNextStep := E_FILE_SCANNER_STEPS.DONE);		
		END_IF	
		
	E_FILE_SCANNER_STEPS.DONE:
		gotoNextStep(iCondition := NOT iScan, iNextStep := E_FILE_SCANNER_STEPS.IDLE);

	E_FILE_SCANNER_STEPS.ERROR:
		oAdsErrorCode := FC_GetAdsErrorCode(scanFolderError);
		gotoNextStep(iCondition := iControlSignals.resetPulse, iNextStep := E_FILE_SCANNER_STEPS.IDLE);
ELSE
	step := E_FILE_SCANNER_STEPS.IDLE;
END_CASE
updateOldStep();


IF (stepChanged AND (step = E_FILE_SCANNER_STEPS.IDLE)) THEN
	fileCnt := 0;
	MEMSET(destAddr := ADR(oFiles), fillByte := 0, SIZEOF(oFiles));
END_IF

IF (stepChanged AND (step = E_FILE_SCANNER_STEPS.SCAN)) THEN
	fileNameAndPath.setPathAndFileName(iPath := iPath, iFileName := iFileName);
	IF (prevStep = E_FILE_SCANNER_STEPS.IDLE) THEN
		fileToSearch := fileNameAndPath.getFileNameNoExtension();

		// Wildcards to find files with similar name
		fileToSearch := FC_3strConcat(iStr1 := fileNameAndPath.getPath(), iStr2 := fileToSearch, iStr3 := IING.STRING_STAR);

		// First scan starts from the beginning (FB_EnumFindFileEntry)
		scanCommand := E_EnumCmdType.eEnumCmd_First;
	ELSE
		// Next scan just continues (FB_EnumFindFileEntry)
		scanCommand := E_EnumCmdType.eEnumCmd_Next;
	END_IF
END_IF

scanFolder(sNetID := iAmsNetId, sPathName := fileToSearch, eCmd := scanCommand, bExecute := (step = E_FILE_SCANNER_STEPS.SCAN), tTimeout := IING.ADS_WRITE_TIMEOUT,
	nErrID => scanFolderError);

oDone := (step = E_FILE_SCANNER_STEPS.DONE);
oFilesFound := fileCnt;
oError := (step = E_FILE_SCANNER_STEPS.ERROR);

METHOD PRIVATE gotoNextStep : BOOL
VAR_INPUT
	iCondition:	BOOL;
	iNextStep:	E_FILE_SCANNER_STEPS;
END_VAR
IF (NOT (step<>oldStepForStepChangeOnly)) THEN
	IF (iCondition) THEN
		step := iNextStep;
	END_IF
END_IF
END_METHOD

ACTION updateOldStep:
IF (step <> oldStepForStepChangeOnly) THEN
	stepChanged := TRUE;
	prevStep := oldStepForStepChangeOnly;			// Otherwise next SWITCH CASE checks oldStep which was just updated here!!
	oldStepForStepChangeOnly := step;
ELSE 
	stepChanged := FALSE;
END_IF
END_ACTION

END_FUNCTION_BLOCK

// ---- LOGGING/Specs/FB_LogLevel.TcPOU
FUNCTION_BLOCK FB_LogLevel		// Helper for setting and getting ENUM as string
VAR
	level:	E_LOG_LEVEL;
END_VAR

METHOD PUBLIC asString : T_DEFAULT_STR
CASE level OF
	E_LOG_LEVEL.TRACE:
		asString := '[TRACE]';
	
	E_LOG_LEVEL.DEBUG:
		asString := '[DEBUG]';
	
	E_LOG_LEVEL.INFO:
		asString := '[INFO]';
	
	E_LOG_LEVEL.WARN:
		asString := '[WARN]';
	
	E_LOG_LEVEL.ERROR:
		asString := '[ERROR]';

	E_LOG_LEVEL.OFF:
		asString := 'do not use this log level';

ELSE
	asString := 'todo';
END_CASE
END_METHOD

METHOD public set : BOOL
VAR_INPUT
	iLevel:	E_LOG_LEVEL;
END_VAR
level := iLevel;
END_METHOD

END_FUNCTION_BLOCK

// ---- LOGGING/GenericLogger/FB_GenericLogger.TcPOU
FUNCTION_BLOCK FB_GenericLogger EXTENDS FB_GenericObserver IMPLEMENTS I_Logger		// Logger where real implementations can subscribe too
																					// This logger by itself does nothing
VAR
	// These VARs cannot be locally inside the METHODs since Twincat does not like that (will crash)
	helperPtr:					POINTER TO BYTE;	// Helper pointer to get the address of the interface
	helperIf:					I_Logger;	// Helper interface for casting back from POINTER TO BOOL to this interface
END_VAR
VAR PERSISTENT
	initCalled: 	INT;
	reInitCalled:	INT;
	exitCalled:		INT;
END_VAR

METHOD PUBLIC debug : BOOL	// Logs the data with log level 'DEBUG'
VAR_INPUT
	iData:		T_DEFAULT_STR;						// Data to be logged, limited to 255 characters
END_VAR
VAR
	i:				INT;
END_VAR
getObservers();
FOR i := 0 TO validObservers.cnt -1 BY 1 DO
	MEMCPY(ADR(helperIf), ADR(validObservers.observers[i].observer), 16);
	helperIf.debug(iData);
END_FOR
END_METHOD

METHOD PUBLIC deregister : BOOL
VAR_INPUT
	iWho:				T_SHORT_STR;
END_VAR
deregisterObserver(iWho);
END_METHOD

METHOD PUBLIC doLog : BOOL	// Logs the data with log level 'WARN'
VAR_INPUT
	iData:		T_DEFAULT_STR;						// Data to be logged, limited to 255 characters
	iLevel:		E_LOG_LEVEL := E_LOG_LEVEL.ERROR;	// Log level
END_VAR
VAR
	i:				INT;
END_VAR
getObservers();
FOR i := 0 TO validObservers.cnt -1 BY 1 DO
	MEMCPY(ADR(helperIf), ADR(validObservers.observers[i].observer), 16);
	helperIf.doLog(iData, iLevel);
END_FOR
END_METHOD

METHOD PUBLIC error : BOOL	// Logs the data with log level 'ERROR'
VAR_INPUT
	iData:		T_DEFAULT_STR;						// Data to be logged, limited to 255 characters
END_VAR
VAR
	i:				INT;
END_VAR
getObservers();
FOR i := 0 TO validObservers.cnt -1 BY 1 DO
	MEMCPY(ADR(helperIf), ADR(validObservers.observers[i].observer), 16);
	helperIf.error(iData);
END_FOR
END_METHOD

METHOD FB_exit : BOOL
VAR_INPUT
	bInCopyCode : BOOL; // if TRUE, the exit method is called for exiting an instance that is copied afterwards (online change).
END_VAR
IncInt(exitCalled);
END_METHOD

METHOD FB_init : BOOL
VAR_INPUT
	bInitRetains : BOOL; // if TRUE, the retain variables are initialized (warm start / cold start)
	bInCopyCode : BOOL;  // if TRUE, the instance afterwards gets moved into the copy code (online change)
END_VAR
IncInt(initCalled);
END_METHOD

METHOD FB_reinit : BOOL
IncInt(reInitCalled);
END_METHOD

METHOD PUBLIC info : BOOL	// Logs the data with log level 'INFO'
VAR_INPUT
	iData:		T_DEFAULT_STR;						// Data to be logged, limited to 255 characters
END_VAR
VAR
	i:				INT;
END_VAR
getObservers();
FOR i := 0 TO validObservers.cnt -1 BY 1 DO
	MEMCPY(ADR(helperIf), ADR(validObservers.observers[i].observer), 16);
	helperIf.info(iData);
END_FOR
END_METHOD

METHOD PUBLIC register : BOOL
VAR_INPUT
	iWho:		T_SHORT_STR;
	iObserver:	I_Logger;
END_VAR
VAR
	pointerSize:	UINT;
END_VAR
// Get the pointer value from the observer Interface

pointerSize := SIZEOF(helperPtr);
MEMCPY(ADR(helperPtr), ADR(iObserver), pointerSize);

registerObserver(iWho, helperPtr);
END_METHOD

METHOD PUBLIC trace : BOOL	// Logs the data with log level 'TRACE'
VAR_INPUT
	iData:		T_DEFAULT_STR;						// Data to be logged, limited to 255 characters
END_VAR
VAR
	i:				INT;
END_VAR
getObservers();
FOR i := 0 TO validObservers.cnt -1 BY 1 DO
	MEMCPY(ADR(helperIf), ADR(validObservers.observers[i].observer), 16);
	helperIf.trace(iData);
END_FOR
END_METHOD

METHOD PUBLIC warn : BOOL	// Logs the data with log level 'WARN'
VAR_INPUT
	iData:		T_DEFAULT_STR;						// Data to be logged, limited to 255 characters
END_VAR
VAR
	i:				INT;
END_VAR
getObservers();
FOR i := 0 TO validObservers.cnt -1 BY 1 DO
	MEMCPY(ADR(helperIf), ADR(validObservers.observers[i].observer), 16);
	helperIf.warn(iData);
END_FOR
END_METHOD

END_FUNCTION_BLOCK

// ---- BASE/AdsUtils/TL_ADS_ERRORS.TcTLO
TEXTLIST TL_ADS_ERRORS
  0 = 'NO_ERROR'
  6 = 'TARGET_PORT_NOT_FOUND'
  7 = 'TARGET_MACHINE_NOT_FOUND'
  1792 = 'ADSERR_DEVICE_ERROR'
  1793 = 'ADSERR_DEVICE_SRVNOTSUPP'
  1794 = 'ADSERR_DEVICE_INVALIDGRP'
  1795 = 'ADSERR_DEVICE_INVALIDOFFSET'
  1796 = 'ADSERR_DEVICE_INVALIDACCESS'
  1797 = 'ADSERR_DEVICE_INVALIDSIZE'
  1798 = 'ADSERR_DEVICE_INVALIDDATA'
  1799 = 'ADSERR_DEVICE_NOTREADY'
  1800 = 'ADSERR_DEVICE_BUSY'
  1801 = 'ADSERR_DEVICE_INVALIDCONTEXT'
  1802 = 'ADSERR_DEVICE_NOMEMORY'
  1803 = 'ADSERR_DEVICE_INVALIDPARM'
  1804 = 'ADSERR_DEVICE_NOTFOUND'
  1805 = 'ADSERR_DEVICE_SYNTAX'
  1806 = 'ADSERR_DEVICE_INCOMPATIBLE'
  1807 = 'ADSERR_DEVICE_EXISTS'
  1808 = 'ADSERR_DEVICE_SYMBOLNOTFOUND'
  1809 = 'ADSERR_DEVICE_SYMBOLVERSIONINVAL'
  1810 = 'ADSERR_DEVICE_INVALIDSTATE'
  1811 = 'ADSERR_DEVICE_TRANSMODENOTSUPP'
  1812 = 'ADSERR_DEVICE_NOTIFYHNDINVALID'
  1813 = 'ADSERR_DEVICE_CLIENTUNKNOWN'
  1814 = 'ADSERR_DEVICE_NOMOREHDLS'
  1815 = 'ADSERR_DEVICE_INVALIDWATCHSIZE'
  1816 = 'ADSERR_DEVICE_NOTINIT'
  1817 = 'ADSERR_DEVICE_TIMEOUT'
  1818 = 'ADSERR_DEVICE_NOINTERFACE'
  1819 = 'ADSERR_DEVICE_INVALIDINTERFACE'
  1820 = 'ADSERR_DEVICE_INVALIDCLSID'
  1821 = 'ADSERR_DEVICE_INVALIDOBJID'
  1822 = 'ADSERR_DEVICE_PENDING'
  1823 = 'ADSERR_DEVICE_ABORTED'
  1824 = 'ADSERR_DEVICE_WARNING'
  1825 = 'ADSERR_DEVICE_INVALIDARRAYIDX'
  1826 = 'ADSERR_DEVICE_SYMBOLNOTACTIVE'
  1827 = 'ADSERR_DEVICE_ACCESSDENIED'
  1828 = 'ADSERR_DEVICE_LICENSENOTFOUND'
  1829 = 'ADSERR_DEVICE_LICENSEEXPIRED'
  1830 = 'ADSERR_DEVICE_LICENSEEXCEEDED'
  1831 = 'ADSERR_DEVICE_LICENSEINVALID'
  1832 = 'ADSERR_DEVICE_LICENSESYSTEMID'
  1833 = 'ADSERR_DEVICE_LICENSENOTIMELIMIT'
  1834 = 'ADSERR_DEVICE_LICENSEFUTUREISSUE'
  1835 = 'ADSERR_DEVICE_LICENSETIMETOLONG'
  1836 = 'ADSERR_DEVICE_EXCEPTION'
  1837 = 'ADSERR_DEVICE_LICENSEDUPLICATED'
  1838 = 'ADSERR_DEVICE_SIGNATUREINVALID'
  1839 = 'ADSERR_DEVICE_CERTIFICATEINVALID'
  1856 = 'ADSERR_CLIENT_ERROR'
  1857 = 'ADSERR_CLIENT_INVALIDPARM'
  1858 = 'ADSERR_CLIENT_LISTEMPTY'
  1859 = 'ADSERR_CLIENT_VARUSED'
  1860 = 'ADSERR_CLIENT_DUPLINVOKEID'
  1861 = 'ADSERR_CLIENT_SYNCTIMEOUT'
  1862 = 'ADSERR_CLIENT_W32ERROR'
  1863 = 'ADSERR_CLIENT_TIMEOUTINVALID'
  1864 = 'ADSERR_CLIENT_PORTNOTOPEN'
  1872 = 'ADSERR_CLIENT_NOAMSADDR'
  1873 = 'ADSERR_CLIENT_SYNCINTERNAL'
  1874 = 'ADSERR_CLIENT_ADDHASH'
  1875 = 'ADSERR_CLIENT_REMOVEHASH'
  1876 = 'ADSERR_CLIENT_NOMORESYM'
  1877 = 'ADSERR_CLIENT_SYNCRESINVALID'
  9999 = 'TODO'
   = ''
END_TEXTLIST

// ---- LOGGING/Specs/TL_LOG_LEVEL.TcTLO
TEXTLIST TL_LOG_LEVEL
  0 = 'TRACE'
  1 = 'DEBUG'
  2 = 'INFO'
  3 = 'WARN'
  4 = 'ERROR'
  5 = 'OFF'
   = ''
END_TEXTLIST
